PROGRAM P20_BackgroundCom
VAR
END_VAR

(* background communication with the EL6031 terminal to *)
// Thermal Bath x 6
// Line Heat x 8
P21_Background_LineHeater();
P22_Background_ThermalBath();

END_PROGRAM

(* stored: Version 1.1.0.1, ProductVersion 3.1.4024.12
   POU P20_BackgroundCom: Id {e6b0834e-6af3-41cd-a374-5856d6875f1e}, SpecialFunc None *)
